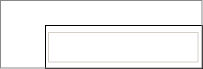
VISUALIZATION Vis_AnalogueOutput_Symbol  // 203x69
VAR_IN_OUT
	stHMI_AnalogueOutput:stHMI_AnalogueOutput;;
END_VAR
    Rectangle (45,25 158x44), colour toggle: NOT(stHMI_AnalogueOutput.bInterlock)
    Textfield (48,32 150x30), text variable: stHMI_AnalogueOutput.rValue
END_VISUALIZATION

(* stored: Version 1.1.0.1, ProductVersion 3.1.4024.11
   Visu Vis_AnalogueOutput_Symbol: Id {b0742e59-2e7c-4822-9865-a0275d210e5e} *)
